// TIA Portal V20 export
FUNCTION_BLOCK "LER_ServoTorqueCal"   // FB20, LAD
// stored: Access Published, MemoryReserve 100, SetENOAutomatically false
   VAR_INPUT
      enable : Bool;
      enableManualCmds : Bool;
      storageCount : UInt;
      storageCycle : Bool;
      RatedTorque : LReal;
      axis : DB_ANY;
   END_VAR
   VAR_OUTPUT
      actualTorque : LReal;
      averageTorque : LReal;
      peakTorque : LReal;
      currentload : LReal;
      averageload : LReal;
      peakload : LReal;
   END_VAR
   VAR_IN_OUT
      configuration : "LER_typeServoTorqueCalConfigruation";
      controlNode : "LER_typeServoTorqueCalControlNode";
      moduleInterface : "LER_typeServoTorqueCalInterface";
   END_VAR
   VAR
      statResetCmd : Bool;
      statActualTorque : LReal;
      statAverageTorque : LReal;
      statPeakTorque : LReal;
      statActualLoad : LReal;
      statAverageLoad : LReal;
      statPeakLoad : LReal;
      statCurrentTorqueDataBuf : Array[0..99] of LReal;
      statMoveCount : UInt;
      statOverloadWarning : Bool;
      statOverloadAlarm : Bool;
      statTonTimer : Array[0..9] of TON_TIME;
      statPulse { S7_SetPoint := 'True'} : Array[0..9] of Bool;
   END_VAR
   VAR_TEMP
      tempRefSpeedAxis : REF_TO TO_SpeedAxis;
      tempRefPosAxis : REF_TO TO_PositioningAxis;
      tempRefSyncAxis : REF_TO TO_SynchronousAxis;
      tempIndex : UInt;
      tempCurrentTorqueSum : LReal;
      tempMonitoringCurrentValue : Bool;
      tempMonitoringPeakValue : Bool;
   END_VAR
   VAR_TEMP   // added for the SCL form of the ladder/FBD networks
      _w1 : Bool;
   END_VAR
BEGIN

REGION Network 1 (SCL): Axis Config
   // Check the axis type
   #tempRefSyncAxis ?= #axis;
   #tempRefPosAxis ?= #axis;
   #tempRefSpeedAxis ?= #axis;

   // Torque Data Move
   IF (#tempRefSyncAxis <> NULL) THEN
       //Axis type TOSynch. Axis
       #statActualTorque := #tempRefSyncAxis^.StatusTorqueData.ActualTorque;

   ELSIF (#tempRefPosAxis <> NULL) THEN
       //Axis type is TO_PositioningAxis 
       #statActualTorque := #tempRefPosAxis^.StatusTorqueData.ActualTorque;

   ELSIF (#tempRefSpeedAxis <> NULL) THEN
       //Axis type TO_Speed. Axis
       #statActualTorque := #tempRefSpeedAxis^.StatusTorqueData.ActualTorque;
   END_IF;

   // Move Count
   IF #storageCount <> 0 THEN
       #statMoveCount := #storageCount - 1;

   ELSIF #storageCount = 0 THEN
       #statMoveCount := 1;
   END_IF;
END_REGION

REGION Network 2 (SCL): Input Mapping
   // Reset
   IF #enableManualCmds THEN
       #statResetCmd := #moduleInterface.commands.Reset;
   ELSE
       #statResetCmd := #controlNode.commands.Reset;
   END_IF;


   // Save
   IF #enableManualCmds AND #moduleInterface.commands.Save THEN
       #moduleInterface.monitoring.OverLoad_Warning_SV := #moduleInterface.configuration.OverLoad_Warning_SV;
       #moduleInterface.monitoring.OverLoad_Alarm_SV := #moduleInterface.configuration.OverLoad_Alarm_SV;
   END_IF;
END_REGION

REGION Network 3: Actual Torque Nm to Actual Load %
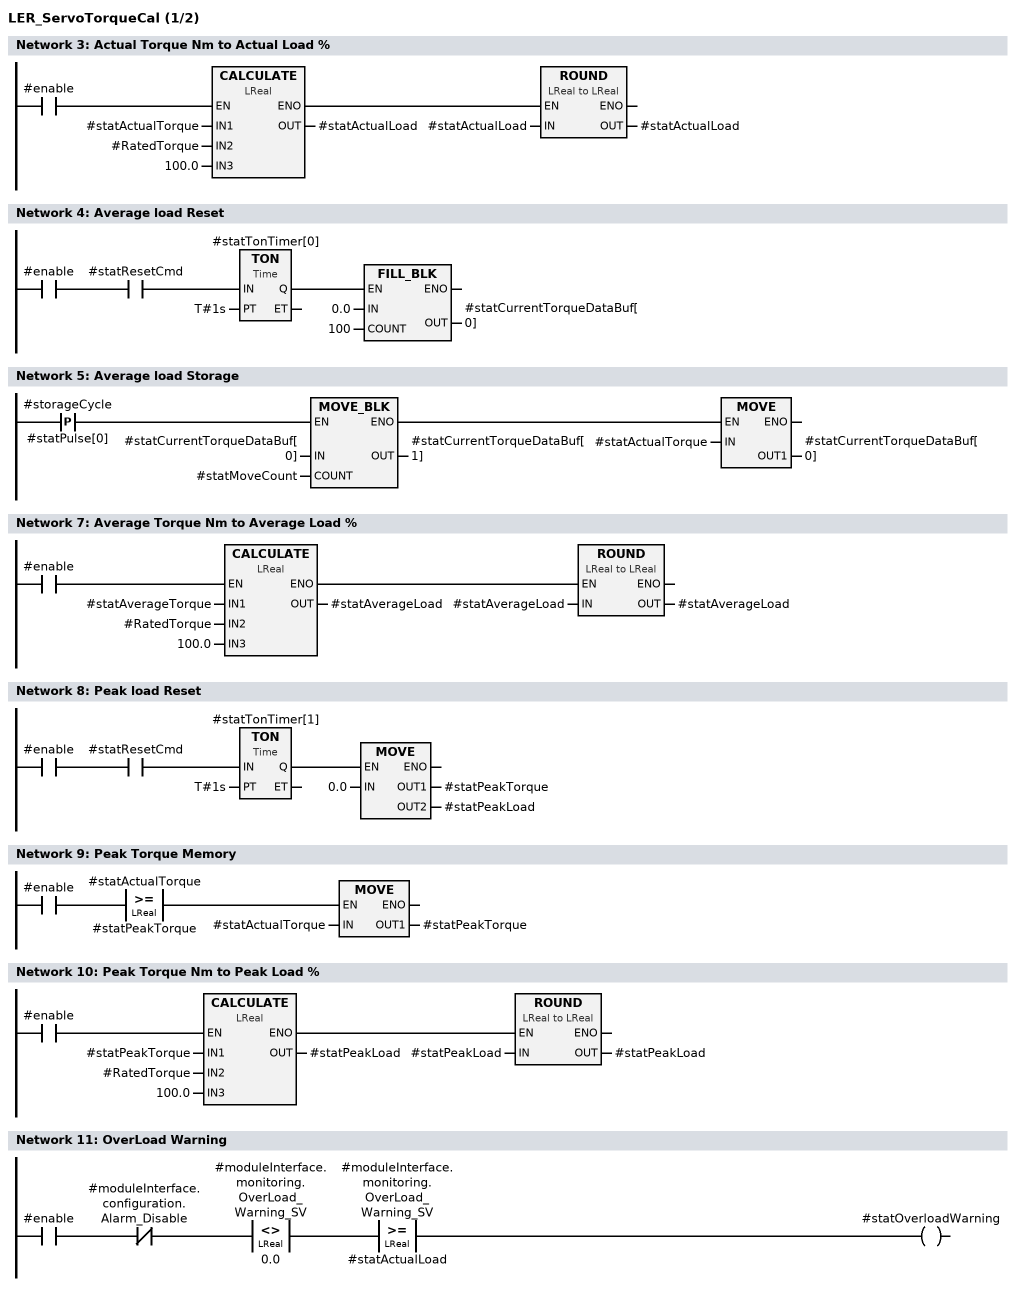
   RUNG wire#powerrail
      Contact( #enable )
      { S7_Templates := "SrcType := LReal"; S7_Expression := "(IN1/IN2)*IN3" } Calculate(in1 := #statActualTorque, in2 := #RatedTorque, in3 := 100.0, out => #statActualLoad)
      { S7_Templates := "[SrcType := LReal, DestType := LReal]" } Round(in := #statActualLoad, out => #statActualLoad)
   END_RUNG
   // the same network as SCL:
   IF #enable THEN
       #statActualLoad := (#statActualTorque/#RatedTorque)*100.0;
       #statActualLoad := ROUND(#statActualLoad);
   END_IF;
END_REGION

REGION Network 4: Average load Reset
   RUNG wire#powerrail
      Contact( #enable )
      Contact( #statResetCmd )
      { S7_Templates := "time_type := Time" } #statTonTimer[0].TON(pt := T#1s, et =>)
      FillBlockI(in := 0.0, count := 100, out => #statCurrentTorqueDataBuf[0])
   END_RUNG
   // the same network as SCL:
   #statTonTimer[0].TON(IN := #enable AND #statResetCmd, PT := T#1s);
   IF #statTonTimer[0].Q THEN FILL_BLK(IN := 0.0, COUNT := 100, OUT => #statCurrentTorqueDataBuf[0]); END_IF;
END_REGION

REGION Network 5: Average load Storage
   // ENO of a box is taken as its EN; it also drops when the box reports an error
   #_w1 := #storageCycle AND NOT #statPulse[0];   // rising edge of #storageCycle
   #statPulse[0] := #storageCycle;
   IF #_w1 THEN
       MOVE_BLK(IN := #statCurrentTorqueDataBuf[0], COUNT := #statMoveCount, OUT => #statCurrentTorqueDataBuf[1]);
       #statCurrentTorqueDataBuf[0] := #statActualTorque;
   END_IF;
END_REGION

REGION Network 6 (SCL): Average Torque Valve
   IF #enable THEN // Current Load Percent Average
       IF #storageCount > 0 THEN
           FOR #tempIndex := 0 TO #storageCount BY 1 DO
               #tempCurrentTorqueSum := #statCurrentTorqueDataBuf[#tempIndex] + #tempCurrentTorqueSum;
           END_FOR;
           #statAverageTorque := #tempCurrentTorqueSum / #storageCount;
       END_IF;
   END_IF;
END_REGION

REGION Network 7: Average Torque Nm to Average Load %
   RUNG wire#powerrail
      Contact( #enable )
      { S7_Templates := "SrcType := LReal"; S7_Expression := "(IN1/IN2)*IN3" } Calculate(in1 := #statAverageTorque, in2 := #RatedTorque, in3 := 100.0, out => #statAverageLoad)
      { S7_Templates := "[SrcType := LReal, DestType := LReal]" } Round(in := #statAverageLoad, out => #statAverageLoad)
   END_RUNG
   // the same network as SCL:
   IF #enable THEN
       #statAverageLoad := (#statAverageTorque/#RatedTorque)*100.0;
       #statAverageLoad := ROUND(#statAverageLoad);
   END_IF;
END_REGION

REGION Network 8: Peak load Reset
   RUNG wire#powerrail
      Contact( #enable )
      Contact( #statResetCmd )
      { S7_Templates := "time_type := Time" } #statTonTimer[1].TON(pt := T#1s, et =>)
      Move(in := 0.0, out1 => #statPeakTorque, out2 => #statPeakLoad)
   END_RUNG
   // the same network as SCL:
   #statTonTimer[1].TON(IN := #enable AND #statResetCmd, PT := T#1s);
   IF #statTonTimer[1].Q THEN
       #statPeakTorque := 0.0;
       #statPeakLoad := 0.0;
   END_IF;
END_REGION

REGION Network 9: Peak Torque Memory
   RUNG wire#powerrail
      Contact( #enable )
      { S7_Templates := "SrcType := LReal" } GE_Contact(in1 := #statActualTorque, in2 := #statPeakTorque)
      Move(in := #statActualTorque, out1 => #statPeakTorque)
   END_RUNG
   // the same network as SCL:
   IF #enable AND (#statActualTorque >= #statPeakTorque) THEN #statPeakTorque := #statActualTorque; END_IF;
END_REGION

REGION Network 10: Peak Torque Nm to Peak Load %
   RUNG wire#powerrail
      Contact( #enable )
      { S7_Templates := "SrcType := LReal"; S7_Expression := "(IN1/IN2)*IN3" } Calculate(in1 := #statPeakTorque, in2 := #RatedTorque, in3 := 100.0, out => #statPeakLoad)
      { S7_Templates := "[SrcType := LReal, DestType := LReal]" } Round(in := #statPeakLoad, out => #statPeakLoad)
   END_RUNG
   // the same network as SCL:
   IF #enable THEN
       #statPeakLoad := (#statPeakTorque/#RatedTorque)*100.0;
       #statPeakLoad := ROUND(#statPeakLoad);
   END_IF;
END_REGION

REGION Network 11: OverLoad Warning
   RUNG wire#powerrail
      Contact( #enable )
      I_Contact( #moduleInterface.configuration.Alarm_Disable )
      { S7_Templates := "SrcType := LReal" } NE_Contact(in1 := #moduleInterface.monitoring.OverLoad_Warning_SV, in2 := 0.0)
      { S7_Templates := "SrcType := LReal" } GE_Contact(in1 := #moduleInterface.monitoring.OverLoad_Warning_SV, in2 := #statActualLoad)
      Coil( #statOverloadWarning )
   END_RUNG
   // the same network as SCL:
   #statOverloadWarning := #enable AND NOT #moduleInterface.configuration.Alarm_Disable AND (#moduleInterface.monitoring.OverLoad_Warning_SV <> 0.0) AND (#moduleInterface.monitoring.OverLoad_Warning_SV >= #statActualLoad);
END_REGION

REGION Network 12: OverLoad Alarm
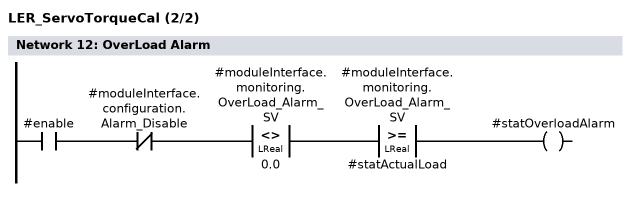
   RUNG wire#powerrail
      Contact( #enable )
      I_Contact( #moduleInterface.configuration.Alarm_Disable )
      { S7_Templates := "SrcType := LReal" } NE_Contact(in1 := #moduleInterface.monitoring.OverLoad_Alarm_SV, in2 := 0.0)
      { S7_Templates := "SrcType := LReal" } GE_Contact(in1 := #moduleInterface.monitoring.OverLoad_Alarm_SV, in2 := #statActualLoad)
      Coil( #statOverloadAlarm )
   END_RUNG
   // the same network as SCL:
   #statOverloadAlarm := #enable AND NOT #moduleInterface.configuration.Alarm_Disable AND (#moduleInterface.monitoring.OverLoad_Alarm_SV <> 0.0) AND (#moduleInterface.monitoring.OverLoad_Alarm_SV >= #statActualLoad);
END_REGION

REGION Network 13 (SCL): OutputMapping
   #moduleInterface.monitoring.OverLoad_Warning := #statOverloadWarning;
   #moduleInterface.monitoring.OverLoad_Alarm := #statOverloadAlarm;

   #moduleInterface.monitoring.Actual_Torque := #actualTorque := #statActualTorque;
   #moduleInterface.monitoring.Average_Torque := #averageTorque := #statAverageTorque;
   #moduleInterface.monitoring.Peak_Torque := #peakTorque := #statPeakTorque;

   #moduleInterface.monitoring.Current_load := #currentload := #statActualLoad;
   #moduleInterface.monitoring.Average_load := #averageload := #statAverageLoad;
   #moduleInterface.monitoring.Peak_load := #peakload := #statPeakLoad;

   #controlNode.monitoring := #moduleInterface.monitoring;
END_REGION
END_FUNCTION_BLOCK
